ORGANIZATION_BLOCK MAIN:OB1
TITLE=H2O2 Control System
BEGIN
Network 1
LD     SM0.1
MOVB   0, VB100
MOVB   0, VB101
R      Q0.0, 8
R      Q1.0, 1
R      M0.0, 2
MOVW   13824, VW1120
MOVW   13824, VW1122
MOVW   0, VW1200
MOVW   0, VW1202
MOVW   0, VW1204
MOVW   0, VW1206

Network 2
LD     I0.3
MOVB   0, VB100
MOVB   0, VB101
R      Q0.0, 8
R      Q1.0, 1
R      M0.0, 2

Network 3
LD     I0.1
AN     I0.3
AB=    VB100, 0
AB=    VB101, 0
MOVB   10, VB100

Network 4
LD     I0.2
AN     I0.3
MOVB   0, VB100
MOVB   10, VB101

Network 5
LD     SM0.0
MOVW   AIW16, VW1000

Network 6
LD     SM0.0
MOVW   AIW18, VW1002

Network 7
LD     SM0.0
MOVW   AIW20, VW1004

Network 8
LD     SM0.0
MOVW   AIW22, VW1010

Network 9
LD     SM0.0
MOVW   AIW24, VW1012

Network 10
LD     SM0.0
MOVW   AIW26, VW1014

Network 11
LD     SM0.0
MOVW   AIW28, VW1016

Network 12
LD     SM0.0
MOVW   AIW30, VW1018

Network 13
LD     SM0.0
AB=    VB100, 10
S      Q0.7, 1
S      Q0.2, 1
S      Q0.3, 1

Network 14
LD     SM0.0
AB=    VB100, 10
AW>=   VW1002, 100
R      Q0.2, 1

Network 15
LD     SM0.0
AB=    VB100, 10
AW>=   VW1004, 100
R      Q0.3, 1

Network 16
LD     SM0.0
AB=    VB100, 10
AN     Q0.2
AN     Q0.3
MOVB   20, VB100

Network 17
LD     SM0.0
AB=    VB100, 20
S      Q0.6, 1
TON    T37, 30

Network 18
LD     SM0.0
AB=    VB100, 20
A      T37
MOVB   30, VB100

Network 19
LD     SM0.0
AB=    VB100, 30
S      Q0.4, 1
TON    T38, 30

Network 20
LD     SM0.0
AB=    VB100, 30
A      T38
MOVB   40, VB100

Network 21
LD     SM0.0
AB=    VB100, 40
S      M0.0, 1

Network 22
LD     SM0.0
AB=    VB100, 40
AW>=   VW1000, 1000
MOVB   50, VB100

Network 23
LD     SM0.0
AB=    VB100, 50
S      M0.1, 1
TON    T39, 30

Network 24
LD     SM0.0
AB=    VB100, 50
A      T39
MOVB   60, VB100

Network 25
LD     SM0.0
AB=    VB100, 60
S      Q0.5, 1
TON    T40, 3000

Network 26
LD     SM0.0
AB=    VB100, 60
A      T40
MOVB   70, VB100

Network 27
LD     SM0.0
AB=    VB100, 70
S      Q1.0, 1
MOVB   100, VB100

Network 28
LD     SM0.0
AB=    VB101, 10
R      Q1.0, 1
R      Q0.2, 2
R      Q0.7, 1
R      M0.1, 1
R      Q0.5, 1
R      M0.0, 1
R      Q0.4, 1
MOVB   20, VB101

Network 29
LD     SM0.0
AB=    VB101, 20
TON    T41, 18000

Network 30
LD     M0.0
MOVW   VW1120, AQW32

Network 31
LD     SM0.0
AN     M0.0
MOVW   0, AQW32

Network 32
LD     M0.1
MOVW   VW1122, AQW34

Network 33
LD     SM0.0
AN     M0.1
MOVW   0, AQW34

Network 34
LD     SM0.1
MOVB   16#F8, SMB37
MOVW   0, SMW38
MOVW   0, SMW42
HDEF   0, 0
HSC    0

Network 35
LD     SM0.1
MOVB   16#F8, SMB47
MOVW   0, SMW48
MOVW   0, SMW52
HDEF   1, 0
HSC    1

Network 36
LD     SM0.0
TON    T42, 100

Network 37
LD     T42
MOVW   SMW38, VW1206
MOVW   SMW48, VW1202

Network 38
LD     T42
AW>=   VW1206, VW1204
SUBW   VW1206, VW1204, VW1200

Network 39
LD     T42
AW<    VW1206, VW1204
MOVW   VW1206, VW1200

Network 40
LD     T42
MOVW   SMW38, VW1204

Network 41
LD     SM0.0
AW>=   VW1200, 1
MOVW   27, VW1210

Network 42
LD     SM0.0
AW>=   VW1200, 2
MOVW   54, VW1210

Network 43
LD     SM0.0
AW>=   VW1200, 3
MOVW   81, VW1210

Network 44
LD     SM0.0
AW>=   VW1200, 4
MOVW   108, VW1210

Network 45
LD     SM0.0
AW>=   VW1200, 5
MOVW   135, VW1210

Network 46
LD     SM0.0
AW>=   VW1200, 6
MOVW   162, VW1210

Network 47
LD     SM0.0
AW>=   VW1200, 7
MOVW   189, VW1210

Network 48
LD     SM0.0
AW>=   VW1200, 8
MOVW   216, VW1210

Network 49
LD     SM0.0
AW>=   VW1200, 9
MOVW   243, VW1210

Network 50
LD     SM0.0
AW>=   VW1200, 10
MOVW   270, VW1210

Network 51
LD     SM0.0
AW>=   VW1200, 11
MOVW   297, VW1210

Network 52
LD     SM0.0
AW>=   VW1200, 12
MOVW   324, VW1210

Network 53
LD     SM0.0
AW>=   VW1200, 13
MOVW   351, VW1210

Network 54
LD     SM0.0
AW>=   VW1200, 14
MOVW   378, VW1210

Network 55
LD     SM0.0
AW>=   VW1200, 15
MOVW   405, VW1210

Network 56
LD     SM0.0
AW>=   VW1200, 16
MOVW   432, VW1210

Network 57
LD     SM0.0
AW>=   VW1200, 17
MOVW   459, VW1210

Network 58
LD     SM0.0
AW>=   VW1200, 18
MOVW   486, VW1210

Network 59
LD     SM0.0
AW>=   VW1200, 19
MOVW   513, VW1210

Network 60
LD     SM0.0
AW>=   VW1200, 20
MOVW   540, VW1210

Network 61
LD     SM0.0
AW>=   VW1200, 21
MOVW   567, VW1210

Network 62
LD     SM0.0
AW>=   VW1200, 22
MOVW   594, VW1210

Network 63
LD     SM0.0
AW>=   VW1200, 23
MOVW   621, VW1210

Network 64
LD     SM0.0
AW>=   VW1200, 24
MOVW   648, VW1210

Network 65
LD     SM0.0
AW>=   VW1200, 25
MOVW   675, VW1210

Network 66
LD     SM0.0
AW>=   VW1200, 26
MOVW   702, VW1210

Network 67
LD     SM0.0
AW>=   VW1200, 27
MOVW   729, VW1210

Network 68
LD     SM0.0
AW>=   VW1200, 28
MOVW   756, VW1210

Network 69
LD     SM0.0
AW>=   VW1200, 29
MOVW   783, VW1210

Network 70
LD     SM0.0
AW>=   VW1200, 30
MOVW   810, VW1210

Network 71
LD     SM0.0
AW>=   VW1202, 1
MOVW   27, VW1212

Network 72
LD     SM0.0
AW>=   VW1202, 2
MOVW   54, VW1212

Network 73
LD     SM0.0
AW>=   VW1202, 3
MOVW   81, VW1212

Network 74
LD     SM0.0
AW>=   VW1202, 4
MOVW   108, VW1212

Network 75
LD     SM0.0
AW>=   VW1202, 5
MOVW   135, VW1212

Network 76
LD     SM0.0
AW>=   VW1202, 6
MOVW   162, VW1212

Network 77
LD     SM0.0
AW>=   VW1202, 7
MOVW   189, VW1212

Network 78
LD     SM0.0
AW>=   VW1202, 8
MOVW   216, VW1212

Network 79
LD     SM0.0
AW>=   VW1202, 9
MOVW   243, VW1212

Network 80
LD     SM0.0
AW>=   VW1202, 10
MOVW   270, VW1212

Network 81
LD     SM0.0
AW>=   VW1202, 11
MOVW   297, VW1212

Network 82
LD     SM0.0
AW>=   VW1202, 12
MOVW   324, VW1212

Network 83
LD     SM0.0
AW>=   VW1202, 13
MOVW   351, VW1212

Network 84
LD     SM0.0
AW>=   VW1202, 14
MOVW   378, VW1212

Network 85
LD     SM0.0
AW>=   VW1202, 15
MOVW   405, VW1212

Network 86
LD     SM0.0
AW>=   VW1202, 16
MOVW   432, VW1212

Network 87
LD     SM0.0
AW>=   VW1202, 17
MOVW   459, VW1212

Network 88
LD     SM0.0
AW>=   VW1202, 18
MOVW   486, VW1212

Network 89
LD     SM0.0
AW>=   VW1202, 19
MOVW   513, VW1212

Network 90
LD     SM0.0
AW>=   VW1202, 20
MOVW   540, VW1212

Network 91
LD     SM0.0
AW>=   VW1202, 21
MOVW   567, VW1212

Network 92
LD     SM0.0
AW>=   VW1202, 22
MOVW   594, VW1212

Network 93
LD     SM0.0
AW>=   VW1202, 23
MOVW   621, VW1212

Network 94
LD     SM0.0
AW>=   VW1202, 24
MOVW   648, VW1212

Network 95
LD     SM0.0
AW>=   VW1202, 25
MOVW   675, VW1212

Network 96
LD     SM0.0
AW>=   VW1202, 26
MOVW   702, VW1212

Network 97
LD     SM0.0
AW>=   VW1202, 27
MOVW   729, VW1212

Network 98
LD     SM0.0
AW>=   VW1202, 28
MOVW   756, VW1212

Network 99
LD     SM0.0
AW>=   VW1202, 29
MOVW   783, VW1212

Network 100
LD     SM0.0
AW>=   VW1202, 30
MOVW   810, VW1212

END_ORGANIZATION_BLOCK
